SUBAPPLICATION Uebung_073d_AUI (* VDS auf UT ausgeben mit AR_Timeout_Zero (Adapter Version) *)
  (* Standard: 61499-2; Description: Copyright (c) 2026 Meisterschulen am Ostbahnhof This program and the accompanying materials are made available under the terms of the Eclipse Public License 2.0 which is available at https://www.eclipse.org/legal/epl-2.0/ SPDX-License-Identifier: EPL-2.0 *)
  (* Version 1.0, 2026-09-17, Franz Höpfinger, Meisterschulen am Ostbahnhof, VDS (Navigation-Based Vehicle Speed) mit PHYS Skalierung und AR_Timeout_Zero Fendt-Schaltung (Adapter Version, analog Krauternter TECU_VDS.SUB) *)
  PACKAGE Uebungen;
  IMPORT Uebungen::const::UT::TECU::DefaultPool_TECU_Numeric::NumberVariable_Ground_based_machine_speed_N;
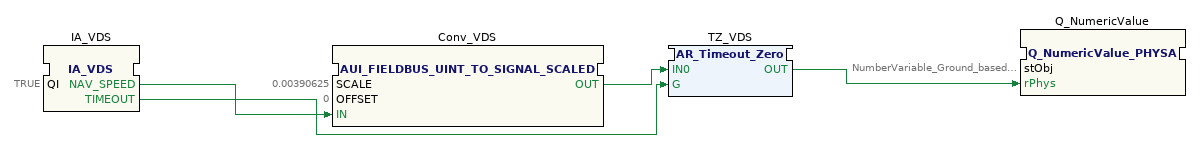
  FBS
    IA_VDS : isobus::tecu::IA_VDS(QI := TRUE);
    Conv_VDS : logiBUS::signalprocessing::fieldbus::AUI_FIELDBUS_UINT_TO_SIGNAL_SCALED(SCALE := 0.00390625, OFFSET := 0);
    Q_NumericValue : isobus::UT::Q::Q_NumericValue_PHYSA(stObj := NumberVariable_Ground_based_machine_speed_N);
  END_FBS
  SUBAPPS
    TZ_VDS : MyLib::sys::AR_Timeout_Zero;
  END_SUBAPPS
  ADAPTER_CONNECTIONS
    IA_VDS.NAV_SPEED TO Conv_VDS.IN;
    Conv_VDS.OUT TO TZ_VDS.IN0;
    IA_VDS.TIMEOUT TO TZ_VDS.G;
    TZ_VDS.OUT TO Q_NumericValue.rPhys;
  END_CONNECTIONS
END_SUBAPPLICATION
